AssertEquals_STRING(
    Expected := expected,
    Actual := actual,
    Message := 'Type did not return correct iec type.'
);

TEST_FINISHED();
END_METHOD

METHOD PUBLIC TestIsSigned
VAR
    _type : _ULINT(0);
    expected : STRING := 'BOOL';
    actual : STRING;
END_VAR
TEST('TestIsSigned');

AssertFalse(
	Condition := _type.IsSigned,
    Message := 'Type did not correctly identify itself as being unsigned'
);

TEST_FINISHED();
END_METHOD

METHOD PUBLIC TestMakeReferenceToFollowsReference
VAR
    _type : _ULINT(0);
	target : ULINT := 0;
    expected : ULINT := 123;
    actual : ULINT;
END_VAR
TEST('TestMakeReferenceToFollowsReference');

_type.MakeReferenceTo(target);
target := 123;

actual := _type.Value;

AssertEquals(
    Expected := expected,
    Actual := actual,
    Message := 'Value did not follow target change'
);

TEST_FINISHED();
END_METHOD

METHOD PUBLIC TestMakeReferenceToUpdatesReference
VAR
    _type : _ULINT(0);
	target : ULINT := 0;
    expected : ULINT := 123;
    actual : ULINT;
END_VAR
TEST('TestMakeReferenceToUpdatesReference');

_type.MakeReferenceTo(target);
_type.Value := 123;

actual := target;

AssertEquals(
    Expected := expected,
    Actual := actual,
    Message := 'Value did not update target'
);

TEST_FINISHED();
END_METHOD

METHOD PUBLIC TestSerializeTypeWith
VAR
    _type : _ULINT(0);
    serializer : JsonSerializer;
    expected : STRING(500) := '{"datatype":"ULINT","lowerBound":0,"upperBound":18446744073709551615,"isSigned":false}';
    actual : STRING(500);
END_VAR
TEST('TestSerializeTypeWith');

serializer.Reset();
_type.SerializeTypeWith(serializer);
serializer.TryGetSerializedData(ADR(actual), SIZEOF(actual));

AssertEquals_STRING(
    Expected := expected,
    Actual := actual,
    Message := 'Serialization of type did not return correct string.'
);

TEST_FINISHED();
END_METHOD

METHOD PUBLIC TestSerializeWith
VAR
    _type : _ULINT(32767);
    serializer : JsonSerializer;
    expected : STRING := '32767';
    actual : STRING(500);
END_VAR
TEST('TestSerializeWith');

serializer.Reset();
_type.SerializeWith(serializer);
serializer.TryGetSerializedData(ADR(actual), SIZEOF(actual));

AssertEquals_STRING(
    Expected := expected,
    Actual := actual,
    Message := 'Serialization of type data did not return correct string.'
);

TEST_FINISHED();
END_METHOD

METHOD PUBLIC TestSize
VAR
    _type : _ULINT(0);
    expected : UDINT := SIZEOF(ULINT);
    actual : UDINT;
END_VAR
TEST('TestSize');

actual := _type.Size;

AssertEquals_UDINT(
    Expected := Expected,
    Actual := actual,
    Message := 'Type did not return the correct size.'
);

TEST_FINISHED();
END_METHOD

METHOD PUBLIC TestTryDeserializeFrom
VAR
    deserializer : JsonDeserializer;
    feedback : DeserializerFeedback;
    json : STRING := '32767';
    _type : _ULINT(0);
    expected : ULINT := 32767;
    actual : ULINT;
 END_VAR
TEST('TestTryDeserializeFrom');

deserializer.Reset();
deserializer.TryLoad(json);
_type.TryDeserializeFrom(Deserializer, Feedback);

actual := _type.Value;

AssertEquals(
    Expected := expected,
    Actual := actual,
    Message := 'Type did not deserialize correctly.'
);

TEST_FINISHED();
END_METHOD

METHOD PUBLIC TestTryMakeReferenceToFollowsReference
VAR
    _type : _ULINT(0);
	target : _ULINT(0);
    expected : ULINT := 123;
    actual : ULINT;
END_VAR
TEST('TestTryMakeReferenceToFollowsReference');

_type.TryMakeReferenceTo(target);
target.Value := 123;

actual := _type.Value;

AssertEquals(
    Expected := expected,
    Actual := actual,
    Message := 'Value did not follow target change'
);

TEST_FINISHED();
END_METHOD

METHOD PUBLIC TestTryMakeReferenceToUpdatesReference
VAR
    _type : _ULINT(0);
	target : _ULINT(0);
    expected : ULINT := 123;
    actual : ULINT;
END_VAR
TEST('TestTryMakeReferenceToUpdatesReference');

_type.TryMakeReferenceTo(target);
_type.Value := 123;

actual := target.Value;

AssertEquals(
    Expected := expected,
    Actual := actual,
    Message := 'Value did not update target'
);

TEST_FINISHED();
END_METHOD

METHOD PUBLIC TestValueReturnsExpectedAfterChange
VAR
    _type : _ULINT(0);
    expected : ULINT := 32767;
    actual : ULINT;
END_VAR
TEST('TestValueReturnsExpectedAfterChange');

_type.Value := 32767;

actual := _type.Value;

AssertEquals(
    Expected := expected,
    Actual := actual,
    Message := 'Expected value not returned after change.'
);

TEST_FINISHED();
END_METHOD

METHOD PUBLIC TestValueReturnsExpectedAfterInit
VAR
    _type : _ULINT(32767);
    expected : ULINT := 32767;
    actual : ULINT;
END_VAR
TEST('TestValueReturnsExpectedAfterInit');

actual := _type.Value;

AssertEquals(
    Expected := expected,
    Actual := actual,
    Message := 'Expected value not returned after Init.'
);

TEST_FINISHED();
END_METHOD

END_FUNCTION_BLOCK

// ---- Tests/Primitives/_REAL_TestSuite.TcPOU
FUNCTION_BLOCK _REAL_TestSuite EXTENDS TcUnit.FB_TestSuite
VAR
END_VAR

TestAddress();
TestClearReference();
TestClone();
TestIecTypeReturnsExpected();
TestIsSigned();
TestMakeReferenceToFollowsReference();
TestMakeReferenceToUpdatesReference();
TestSize();
TestValueReturnsExpectedAfterInit();
TestValueReturnsExpectedAfterChange();
TestSerializeTypeWith();
TestSerializeWith();
TestTryDeserializeFrom();
TestTryMakeReferenceToFollowsReference();
TestTryMakeReferenceToUpdatesReference();

METHOD PUBLIC TestAddress
VAR
    _type : _REAL(0.0);
    notExpected : PVOID := 0;
    actual : PVOID;
END_VAR
TEST('TestAddress');

actual := _type.Address;

AssertFalse(
    Condition := (notExpected = actual),
    Message := 'Type did not return a valid address.'
);

TEST_FINISHED();
END_METHOD

METHOD PUBLIC TestClearReference
VAR
    _type : _REAL(0.0);
	target : REAL := 0.0;
    expected : REAL := 0.0;
    actual : REAL;
END_VAR
TEST('TestClearReference');

_type.MakeReferenceTo(target);
_type.ClearReference();
target := 123.4;

actual := _type.Value;

AssertEquals_REAL(
    Expected := expected,
    Actual := actual,
    Delta := REAL#0.001,
    Message := 'Value did not follow target change'
);

TEST_FINISHED();
END_METHOD

METHOD PUBLIC TestClone
VAR
    _type : _REAL(123.4);
	clone : I_Datatype;
	isValidClone : BOOL;
	compareResult : DINT;
END_VAR
TEST('TestClone');

clone := _type.Clone();

isValidClone := clone <> 0;

IF isValidClone THEN
	compareResult := memcmp(_type.Address, clone.Address, clone.Size);
END_IF

AssertTrue(
	Condition := isValidClone,
	Message := 'Clone did not produce a clone'
);

AssertEquals_DINT(
	Expected := 0,
    Actual := compareResult,
    Message := 'Clone did not return a valid clone.'
);

clone.Dispose();

TEST_FINISHED();
END_METHOD

METHOD PUBLIC TestIecTypeReturnsExpected
VAR
    _type : _REAL(0.0);
    expected : STRING := 'REAL';
    actual : STRING;
END_VAR
TEST('TestIecTypeReturnsExpected');

actual := _type.Datatype;

AssertEquals_STRING(
    Expected := expected,
    Actual := actual,
    Message := 'Type did not return correct iec type.'
);

TEST_FINISHED();
END_METHOD

METHOD PUBLIC TestIsSigned
VAR
    _type : _REAL(0);
    expected : STRING := 'BOOL';
    actual : STRING;
END_VAR
TEST('TestIsSigned');

AssertTrue(
	Condition := _type.IsSigned,
    Message := 'Type did not correctly identify itself as being signed'
);

TEST_FINISHED();
END_METHOD

METHOD PUBLIC TestMakeReferenceToFollowsReference
VAR
    _type : _REAL(0.0);
	target : REAL := 0.0;
    expected : REAL := 123.4;
    actual : REAL;
END_VAR
TEST('TestMakeReferenceToFollowsReference');

_type.MakeReferenceTo(target);
target := 123.4;

actual := _type.Value;

AssertEquals_REAL(
    Expected := expected,
    Actual := actual,
    Delta := REAL#0.001,
    Message := 'Value did not follow target change'
);

TEST_FINISHED();
END_METHOD

METHOD PUBLIC TestMakeReferenceToUpdatesReference
VAR
    _type : _REAL(0.0);
	target : REAL := 0.0;
    expected : REAL := 123.4;
    actual : REAL;
END_VAR
TEST('TestMakeReferenceToUpdatesReference');

_type.MakeReferenceTo(target);
_type.Value := 123.4;

actual := target;

AssertEquals_REAL(
    Expected := expected,
    Actual := actual,
    Delta := REAL#0.001,
    Message := 'Value did not update target'
);

TEST_FINISHED();
END_METHOD

METHOD PUBLIC TestSerializeTypeWith
VAR
    _type : _REAL(0.0);
    serializer : JsonSerializer;
    expected : STRING(500) := '{"datatype":"REAL"}';
    actual : STRING(500);
END_VAR
TEST('TestSerializeTypeWith');

serializer.Reset();
_type.SerializeTypeWith(serializer);
serializer.TryGetSerializedData(ADR(actual), SIZEOF(actual));

AssertEquals_STRING(
    Expected := expected,
    Actual := actual,
    Message := 'Serialization of type did not return correct string.'
);

TEST_FINISHED();
END_METHOD

METHOD PUBLIC TestSerializeWith
VAR
    _type : _REAL(123.4);
    serializer : JsonSerializer;
    expected : STRING := '123.40000152'; // Expected value due to the nature of floating point values defined by IEEE754.
    actual : STRING(500);
END_VAR
TEST('TestSerializeWith');

serializer.Reset();
_type.SerializeWith(serializer);
serializer.TryGetSerializedData(ADR(actual), SIZEOF(actual));

AssertEquals_STRING(
    Expected := expected,
    Actual := actual,
    Message := 'Serialization of type data did not return correct string.'
);

TEST_FINISHED();
END_METHOD

METHOD PUBLIC TestSize
VAR
    _type : _REAL(0.0);
    expected : UDINT := SIZEOF(REAL);
    actual : UDINT;
END_VAR
TEST('TestSize');

actual := _type.Size;

AssertEquals_UDINT(
    Expected := Expected,
    Actual := actual,
    Message := 'Type did not return the correct size.'
);

TEST_FINISHED();
END_METHOD

METHOD PUBLIC TestTryDeserializeFrom
VAR
    deserializer : JsonDeserializer;
    feedback : DeserializerFeedback;
    json : STRING := '123.4';
    _type : _REAL(0.0);
    expected : REAL := 123.4;
    actual : REAL;
 END_VAR
TEST('TestTryDeserializeFrom');

deserializer.Reset();
deserializer.TryLoad(json);
_type.TryDeserializeFrom(Deserializer, Feedback);

actual := _type.Value;

AssertEquals_REAL(
    Expected := expected,
    Actual := actual,
    Delta := REAL#0.001,
    Message := 'Type did not deserialize correctly.'
);

TEST_FINISHED();
END_METHOD

METHOD PUBLIC TestTryMakeReferenceToFollowsReference
VAR
    _type : _REAL(0.0);
	target : _REAL(0.0);
    expected : REAL := 123.4;
    actual : REAL;
END_VAR
TEST('TestTryMakeReferenceToFollowsReference');

_type.TryMakeReferenceTo(target);
target.Value := 123.4;

actual := _type.Value;

AssertEquals_REAL(
    Expected := expected,
    Actual := actual,
    Delta := REAL#0.001,
    Message := 'Value did not follow target change'
);

TEST_FINISHED();
END_METHOD

METHOD PUBLIC TestTryMakeReferenceToUpdatesReference
VAR
    _type : _REAL(0.0);
	target : _REAL(0.0);
    expected : REAL := 123.4;
    actual : REAL;
END_VAR
TEST('TestTryMakeReferenceToUpdatesReference');

_type.TryMakeReferenceTo(target);
_type.Value := 123.4;

actual := target.Value;

AssertEquals_REAL(
    Expected := expected,
    Actual := actual,
    Delta := REAL#0.001,
    Message := 'Value did not update target'
);

TEST_FINISHED();
END_METHOD

METHOD PUBLIC TestValueReturnsExpectedAfterChange
VAR
    _type : _REAL(0.0);
    expected : REAL := 123.4;
    actual : REAL;
END_VAR
TEST('TestValueReturnsExpectedAfterChange');

_type.Value := 123.4;

actual := _type.Value;

AssertEquals_REAL(
    Expected := expected,
    Actual := actual,
    Delta := REAL#0.001,
    Message := 'Expected value not returned after change.'
);

TEST_FINISHED();
END_METHOD

METHOD PUBLIC TestValueReturnsExpectedAfterInit
VAR
    _type : _REAL(123.4);
    expected : REAL := 123.4;
    actual : REAL;
END_VAR
TEST('TestValueReturnsExpectedAfterInit');

actual := _type.Value;

AssertEquals_REAL(
    Expected := expected,
    Actual := actual,
    Delta := REAL#0.001,
    Message := 'Expected value not returned after Init.'
);

TEST_FINISHED();
END_METHOD

END_FUNCTION_BLOCK

// ---- Tests/Primitives/_LREAL_TestSuite.TcPOU
FUNCTION_BLOCK _LREAL_TestSuite EXTENDS TcUnit.FB_TestSuite
VAR
END_VAR

TestAddress();
TestClearReference();
TestClone();
TestIecTypeReturnsExpected();
TestIsSigned();
TestMakeReferenceToFollowsReference();
TestMakeReferenceToUpdatesReference();
TestSize();
TestValueReturnsExpectedAfterInit();
TestValueReturnsExpectedAfterChange();
TestSerializeTypeWith();
TestSerializeWith();
TestTryDeserializeFrom();
TestTryMakeReferenceToFollowsReference();
TestTryMakeReferenceToUpdatesReference();

METHOD PUBLIC TestAddress
VAR
    _type : _LREAL(0.0);
    notExpected : PVOID := 0;
    actual : PVOID;
END_VAR
TEST('TestAddress');

actual := _type.Address;

AssertFalse(
    Condition := (notExpected = actual),
    Message := 'Type did not return a valid address.'
);

TEST_FINISHED();
END_METHOD

METHOD PUBLIC TestClearReference
VAR
    _type : _LREAL(0.0);
	target : LREAL := 0.0;
    expected : LREAL := 0.0;
    actual : LREAL;
END_VAR
TEST('TestClearReference');

_type.MakeReferenceTo(target);
_type.ClearReference();
target := 123.4;

actual := _type.Value;

AssertEquals_LREAL(
    Expected := expected,
    Actual := actual,
    Delta := LREAL#0.001,
    Message := 'Value did not follow target change'
);

TEST_FINISHED();
END_METHOD

METHOD PUBLIC TestClone
VAR
    _type : _LREAL(123.4);
	clone : I_Datatype;
	isValidClone : BOOL;
	compareResult : DINT;
END_VAR
TEST('TestClone');

clone := _type.Clone();

isValidClone := clone <> 0;

IF isValidClone THEN
	compareResult := memcmp(_type.Address, clone.Address, clone.Size);
END_IF

AssertTrue(
	Condition := isValidClone,
	Message := 'Clone did not produce a clone'
);

AssertEquals_DINT(
	Expected := 0,
    Actual := compareResult,
    Message := 'Clone did not return a valid clone.'
);

clone.Dispose();

TEST_FINISHED();
END_METHOD

METHOD PUBLIC TestIecTypeReturnsExpected
VAR
    _type : _LREAL(0.0);
    expected : STRING := 'LREAL';
    actual : STRING;
END_VAR
TEST('TestIecTypeReturnsExpected');

actual := _type.Datatype;

AssertEquals_STRING(
    Expected := expected,
    Actual := actual,
    Message := 'Type did not return correct iec type.'
);

TEST_FINISHED();
END_METHOD

METHOD PUBLIC TestIsSigned
VAR
    _type : _LREAL(0);
    expected : STRING := 'BOOL';
    actual : STRING;
END_VAR
TEST('TestIsSigned');

AssertTrue(
	Condition := _type.IsSigned,
    Message := 'Type did not correctly identify itself as being signed'
);

TEST_FINISHED();
END_METHOD

METHOD PUBLIC TestMakeReferenceToFollowsReference
VAR
    _type : _LREAL(0.0);
	target : LREAL := 0.0;
    expected : LREAL := 123.4;
    actual : LREAL;
END_VAR
TEST('TestMakeReferenceToFollowsReference');

_type.MakeReferenceTo(target);
target := 123.4;

actual := _type.Value;

AssertEquals_LREAL(
    Expected := expected,
    Actual := actual,
    Delta := LREAL#0.001,
    Message := 'Value did not follow target change'
);

TEST_FINISHED();
END_METHOD

METHOD PUBLIC TestMakeReferenceToUpdatesReference
VAR
    _type : _LREAL(0.0);
	target : LREAL := 0.0;
    expected : LREAL := 123.4;
    actual : LREAL;
END_VAR
TEST('TestMakeReferenceToUpdatesReference');

_type.MakeReferenceTo(target);
_type.Value := 123.4;

actual := target;

AssertEquals_LREAL(
    Expected := expected,
    Actual := actual,
    Delta := LREAL#0.001,
    Message := 'Value did not update target'
);

TEST_FINISHED();
END_METHOD

METHOD PUBLIC TestSerializeTypeWith
VAR
    _type : _LREAL(0.0);
    serializer : JsonSerializer;
    expected : STRING(500) := '{"datatype":"LREAL"}';
    actual : STRING(500);
END_VAR
TEST('TestSerializeTypeWith');

serializer.Reset();
_type.SerializeTypeWith(serializer);
serializer.TryGetSerializedData(ADR(actual), SIZEOF(actual));

AssertEquals_STRING(
    Expected := expected,
    Actual := actual,
    Message := 'Serialization of type did not return correct string.'
);

TEST_FINISHED();
END_METHOD

METHOD PUBLIC TestSerializeWith
VAR
    _type : _LREAL(123.4);
    serializer : JsonSerializer;
    expected : STRING := '123.4';
    actual : STRING(500);
END_VAR
TEST('TestSerializeWith');

serializer.Reset();
_type.SerializeWith(serializer);
serializer.TryGetSerializedData(ADR(actual), SIZEOF(actual));

AssertEquals_STRING(
    Expected := expected,
    Actual := actual,
    Message := 'Serialization of type data did not return correct string.'
);

TEST_FINISHED();
END_METHOD

METHOD PUBLIC TestSize
VAR
    _type : _LREAL(0.0);
    expected : UDINT := SIZEOF(LREAL);
    actual : UDINT;
END_VAR
TEST('TestSize');

actual := _type.Size;

AssertEquals_UDINT(
    Expected := Expected,
    Actual := actual,
    Message := 'Type did not return the correct size.'
);

TEST_FINISHED();
END_METHOD

METHOD PUBLIC TestTryDeserializeFrom
VAR
    deserializer : JsonDeserializer;
    feedback : DeserializerFeedback;
    json : STRING := '123.4';
    _type : _LREAL(0.0);
    expected : LREAL := 123.4;
    actual : LREAL;
 END_VAR
TEST('TestTryDeserializeFrom');

deserializer.Reset();
deserializer.TryLoad(json);
_type.TryDeserializeFrom(Deserializer, Feedback);

actual := _type.Value;

AssertEquals_LREAL(
    Expected := expected,
    Actual := actual,
    Delta := LREAL#0.001,
    Message := 'Type did not deserialize correctly.'
);

TEST_FINISHED();
END_METHOD

METHOD PUBLIC TestTryMakeReferenceToFollowsReference
VAR
    _type : _LREAL(0.0);
	target : _LREAL(0.0);
    expected : LREAL := 123.4;
    actual : LREAL;
END_VAR
TEST('TestTryMakeReferenceToFollowsReference');

_type.TryMakeReferenceTo(target);
target.Value := 123.4;

actual := _type.Value;

AssertEquals_LREAL(
    Expected := expected,
    Actual := actual,
    Delta := LREAL#0.001,
    Message := 'Value did not follow target change'
);

TEST_FINISHED();
END_METHOD

METHOD PUBLIC TestTryMakeReferenceToUpdatesReference
VAR
    _type : _LREAL(0.0);
	target : _LREAL(0.0);
    expected : LREAL := 123.4;
    actual : LREAL;
END_VAR
TEST('TestTryMakeReferenceToUpdatesReference');

_type.TryMakeReferenceTo(target);
_type.Value := 123.4;

actual := target.Value;

AssertEquals_LREAL(
    Expected := expected,
    Actual := actual,
    Delta := LREAL#0.001,
    Message := 'Value did not update target'
);

TEST_FINISHED();
END_METHOD

METHOD PUBLIC TestValueReturnsExpectedAfterChange
VAR
    _type : _LREAL(0.0);
    expected : LREAL := 123.4;
    actual : LREAL;
END_VAR
TEST('TestValueReturnsExpectedAfterChange');

_type.Value := 123.4;

actual := _type.Value;

AssertEquals_LREAL(
    Expected := expected,
    Actual := actual,
    Delta := LREAL#0.001,
    Message := 'Expected value not returned after change.'
);

TEST_FINISHED();
END_METHOD

METHOD PUBLIC TestValueReturnsExpectedAfterInit
VAR
    _type : _LREAL(123.4);
    expected : LREAL := 123.4;
    actual : LREAL;
END_VAR
TEST('TestValueReturnsExpectedAfterInit');

actual := _type.Value;

AssertEquals_LREAL(
    Expected := expected,
    Actual := actual,
    Delta := LREAL#0.001,
    Message := 'Expected value not returned after Init.'
);

TEST_FINISHED();
END_METHOD

END_FUNCTION_BLOCK

// ---- Tests/Primitives/_TOD_TestSuite.TcPOU
FUNCTION_BLOCK _TOD_TestSuite EXTENDS TcUnit.FB_TestSuite
VAR
END_VAR

TestAddress();
TestClearReference();
TestClone();
TestIecTypeReturnsExpected();
TestMakeReferenceToFollowsReference();
TestMakeReferenceToUpdatesReference();
TestSize();
TestValueReturnsExpectedAfterInit();
TestValueReturnsExpectedAfterChange();
TestSerializeTypeWith();
TestSerializeWith();
TestTryDeserializeFrom();
TestTryMakeReferenceToFollowsReference();
TestTryMakeReferenceToUpdatesReference();

METHOD PUBLIC TestAddress
VAR
    _type : _TOD(TOD#0:0:0);
    notExpected : PVOID := 0;
    actual : PVOID;
END_VAR
TEST('TestAddress');

actual := _type.Address;

AssertFalse(
    Condition := (notExpected = actual),
    Message := 'Type did not return a valid address.'
);

TEST_FINISHED();
END_METHOD

METHOD PUBLIC TestClearReference
VAR
    _type : _TOD(TOD#0:0:0);
	target : TOD := TOD#0:0:0;
    expected : TOD := TOD#0:0:0;
    actual : TOD;
END_VAR
TEST('TestClearReference');

_type.MakeReferenceTo(target);
_type.ClearReference();
target := TOD#12:34:56.789;

actual := _type.Value;

AssertEquals(
    Expected := expected,
    Actual := actual,
    Message := 'Value did not follow target change'
);

TEST_FINISHED();
END_METHOD

METHOD PUBLIC TestClone
VAR
    _type : _TIME_OF_DAY(TIME_OF_DAY#12:34:56.789);
	clone : I_Datatype;
	isValidClone : BOOL;
	compareResult : DINT;
END_VAR
TEST('TestClone');

clone := _type.Clone();

isValidClone := clone <> 0;

IF isValidClone THEN
	compareResult := memcmp(_type.Address, clone.Address, clone.Size);
END_IF

AssertTrue(
	Condition := isValidClone,
	Message := 'Clone did not produce a clone'
);

AssertEquals_DINT(
	Expected := 0,
    Actual := compareResult,
    Message := 'Clone did not return a valid clone.'
);

clone.Dispose();

TEST_FINISHED();
END_METHOD

METHOD PUBLIC TestIecTypeReturnsExpected
VAR
    _type : _TOD(TOD#0:0:0);
    expected : STRING := 'TOD';
    actual : STRING;
END_VAR
TEST('TestIecTypeReturnsExpected');

actual := _type.Datatype;

AssertEquals_STRING(
    Expected := expected,
    Actual := actual,
    Message := 'Type did not return correct iec type.'
);

TEST_FINISHED();
END_METHOD

METHOD PUBLIC TestMakeReferenceToFollowsReference
VAR
    _type : _TOD(TOD#0:0:0);
	target : TOD := TOD#0:0:0;
    expected : TOD := TOD#12:34:56.789;
    actual : TOD;
END_VAR
TEST('TestMakeReferenceToFollowsReference');

_type.MakeReferenceTo(target);
target := TOD#12:34:56.789;

actual := _type.Value;

AssertEquals_TIME_OF_DAY(
    Expected := expected,
    Actual := actual,
    Message := 'Value did not follow target change'
);

TEST_FINISHED();
END_METHOD

METHOD PUBLIC TestMakeReferenceToUpdatesReference
VAR
    _type : _TOD(TOD#0:0:0);
	target : TOD := TOD#0:0:0;
    expected : TOD := TOD#12:34:56.789;
    actual : TOD;
END_VAR
TEST('TestMakeReferenceToUpdatesReference');

_type.MakeReferenceTo(target);
_type.Value := TOD#12:34:56.789;

actual := target;

AssertEquals_TIME_OF_DAY(
    Expected := expected,
    Actual := actual,
    Message := 'Value did not update target'
);

TEST_FINISHED();
END_METHOD

METHOD PUBLIC TestSerializeTypeWith
VAR
    _type : _TOD(TOD#0:0:0);
    serializer : JsonSerializer;
    expected : STRING := '{"datatype":"TOD"}';
    actual : STRING(500);
END_VAR
TEST('TestSerializeTypeWith');

serializer.Reset();
_type.SerializeTypeWith(serializer);
serializer.TryGetSerializedData(ADR(actual), SIZEOF(actual));

AssertEquals_STRING(
    Expected := expected,
    Actual := actual,
    Message := 'Serialization of type did not return correct string.'
);

TEST_FINISHED();
END_METHOD

METHOD PUBLIC TestSerializeWith
VAR
    _type : _TOD(TOD#12:34:56.789);
    serializer : JsonSerializer;
    expected : STRING := '"TOD#12:34:56.789"';
    actual : STRING(500);
END_VAR
TEST('TestSerializeWith');

serializer.Reset();
_type.SerializeWith(serializer);
serializer.TryGetSerializedData(ADR(actual), SIZEOF(actual));

AssertEquals_STRING(
    Expected := expected,
    Actual := actual,
    Message := 'Serialization of type data did not return correct string.'
);

TEST_FINISHED();
END_METHOD

METHOD PUBLIC TestSize
VAR
    _type : _TOD(TOD#0:0:0);
    expected : UDINT := SIZEOF(TOD);
    actual : UDINT;
END_VAR
TEST('TestSize');

actual := _type.Size;

AssertEquals_UDINT(
    Expected := Expected,
    Actual := actual,
    Message := 'Type did not return the correct size.'
);

TEST_FINISHED();
END_METHOD

METHOD PUBLIC TestTryDeserializeFrom
VAR
    deserializer : JsonDeserializer;
    feedback : DeserializerFeedback;
    json : STRING := '"TOD#12:34:56.789"';
    _type : _TOD(TOD#0:0:0);
    expected : TOD := TOD#12:34:56.789;
    actual : TOD;
 END_VAR
TEST('TestTryDeserializeFrom');

deserializer.Reset();
deserializer.TryLoad(json);
_type.TryDeserializeFrom(Deserializer, Feedback);

actual := _type.Value;

AssertEquals_TIME_OF_DAY(
    Expected := expected,
    Actual := actual,
    Message := 'Type did not deserialize correctly.'
);

TEST_FINISHED();
END_METHOD

METHOD PUBLIC TestTryMakeReferenceToFollowsReference
VAR
    _type : _TOD(TOD#0:0:0);
	target : _TOD(TOD#0:0:0);
    expected : TOD := TOD#12:34:56.789;
    actual : TOD;
END_VAR
TEST('TestTryMakeReferenceToFollowsReference');

_type.TryMakeReferenceTo(target);
target.Value := TOD#12:34:56.789;

actual := _type.Value;

AssertEquals_TIME_OF_DAY(
    Expected := expected,
    Actual := actual,
    Message := 'Value did not follow target change'
);

TEST_FINISHED();
END_METHOD

METHOD PUBLIC TestTryMakeReferenceToUpdatesReference
VAR
    _type : _TOD(TOD#0:0:0);
	target : _TOD(TOD#0:0:0);
    expected : TOD := TOD#12:34:56.789;
    actual : TOD;
END_VAR
TEST('TestTryMakeReferenceToUpdatesReference');

_type.TryMakeReferenceTo(target);
_type.Value := TOD#12:34:56.789;

actual := target.Value;

AssertEquals_TIME_OF_DAY(
    Expected := expected,
    Actual := actual,
    Message := 'Value did not update target'
);

TEST_FINISHED();
END_METHOD

METHOD PUBLIC TestValueReturnsExpectedAfterChange
VAR
    _type : _TOD(TOD#0:0:0);
    expected : TOD := TOD#12:34:56.789;
    actual : TOD;
END_VAR
TEST('TestValueReturnsExpectedAfterChange');

_type.Value := TOD#12:34:56.789;

actual := _type.Value;

AssertEquals_TIME_OF_DAY(
    Expected := expected,
    Actual := actual,
    Message := 'Expected value not returned after change.'
);

TEST_FINISHED();
END_METHOD

METHOD PUBLIC TestValueReturnsExpectedAfterInit
VAR
    _type : _TOD(TOD#12:34:56.789);
    expected : TOD := TOD#12:34:56.789;
    actual : TOD;
END_VAR
TEST('TestValueReturnsExpectedAfterInit');

actual := _type.Value;

AssertEquals_TIME_OF_DAY(
    Expected := expected,
    Actual := actual,
    Message := 'Expected value not returned after Init.'
);

TEST_FINISHED();
END_METHOD

END_FUNCTION_BLOCK

// ---- Tests/Primitives/_TIME_OF_DAY_TestSuite.TcPOU
FUNCTION_BLOCK _TIME_OF_DAY_TestSuite EXTENDS TcUnit.FB_TestSuite
VAR
END_VAR

TestAddress();
TestClearReference();
TestClone();
TestIecTypeReturnsExpected();
TestMakeReferenceToFollowsReference();
TestMakeReferenceToUpdatesReference();
TestSize();
TestValueReturnsExpectedAfterInit();
TestValueReturnsExpectedAfterChange();
TestSerializeTypeWith();
TestSerializeWith();
TestTryDeserializeFrom();
TestTryMakeReferenceToFollowsReference();
TestTryMakeReferenceToUpdatesReference();

METHOD PUBLIC TestAddress
VAR
    _type : _TIME_OF_DAY(TIME_OF_DAY#0:0:0);
    notExpected : PVOID := 0;
    actual : PVOID;
END_VAR
TEST('TestAddress');

actual := _type.Address;

AssertFalse(
    Condition := (notExpected = actual),
    Message := 'Type did not return a valid address.'
);

TEST_FINISHED();
END_METHOD

METHOD PUBLIC TestClearReference
VAR
    _type : _TIME_OF_DAY(TIME_OF_DAY#0:0:0);
	target : TIME_OF_DAY := TIME_OF_DAY#0:0:0;
    expected : TIME_OF_DAY := TIME_OF_DAY#0:0:0;
    actual : TIME_OF_DAY;
END_VAR
TEST('TestClearReference');

_type.MakeReferenceTo(target);
_type.ClearReference();
target := TIME_OF_DAY#12:34:56.789;

actual := _type.Value;

AssertEquals(
    Expected := expected,
    Actual := actual,
    Message := 'Value did not follow target change'
);

TEST_FINISHED();
END_METHOD

METHOD PUBLIC TestClone
VAR
    _type : _TIME_OF_DAY(TIME_OF_DAY#12:34:56.789);
	clone : I_Datatype;
	isValidClone : BOOL;
	compareResult : DINT;
END_VAR
TEST('TestClone');

clone := _type.Clone();

isValidClone := clone <> 0;

IF isValidClone THEN
	compareResult := memcmp(_type.Address, clone.Address, clone.Size);
END_IF

AssertTrue(
	Condition := isValidClone,
	Message := 'Clone did not produce a clone'
);

AssertEquals_DINT(
	Expected := 0,
    Actual := compareResult,
    Message := 'Clone did not return a valid clone.'
);

clone.Dispose();

TEST_FINISHED();
END_METHOD

METHOD PUBLIC TestIecTypeReturnsExpected
VAR
    _type : _TIME_OF_DAY(TIME_OF_DAY#0:0:0);
    expected : STRING := 'TIME_OF_DAY';
    actual : STRING;
END_VAR
TEST('TestIecTypeReturnsExpected');

actual := _type.Datatype;

AssertEquals_STRING(
    Expected := expected,
    Actual := actual,
    Message := 'Type did not return correct iec type.'
);

TEST_FINISHED();
END_METHOD

METHOD PUBLIC TestMakeReferenceToFollowsReference
VAR
    _type : _TIME_OF_DAY(TIME_OF_DAY#0:0:0);
	target : TIME_OF_DAY := TIME_OF_DAY#0:0:0;
    expected : TIME_OF_DAY := TIME_OF_DAY#12:34:56.789;
    actual : TIME_OF_DAY;
END_VAR
TEST('TestMakeReferenceToFollowsReference');

_type.MakeReferenceTo(target);
target := TIME_OF_DAY#12:34:56.789;;

actual := _type.Value;

AssertEquals_TIME_OF_DAY(
    Expected := expected,
    Actual := actual,
    Message := 'Value did not follow target change'
);

TEST_FINISHED();
END_METHOD

METHOD PUBLIC TestMakeReferenceToUpdatesReference
VAR
    _type : _TIME_OF_DAY(TIME_OF_DAY#0:0:0);
	target : TIME_OF_DAY := TIME_OF_DAY#0:0:0;
    expected : TIME_OF_DAY := TIME_OF_DAY#12:34:56.789;
    actual : TIME_OF_DAY;
END_VAR
TEST('TestMakeReferenceToUpdatesReference');

_type.MakeReferenceTo(target);
_type.Value := TIME_OF_DAY#12:34:56.789;

actual := target;

AssertEquals_TIME_OF_DAY(
    Expected := expected,
    Actual := actual,
    Message := 'Value did not update target'
);

TEST_FINISHED();
END_METHOD

METHOD PUBLIC TestSerializeTypeWith
VAR
    _type : _TIME_OF_DAY(TIME_OF_DAY#0:0:0);
    serializer : JsonSerializer;
    expected : STRING := '{"datatype":"TIME_OF_DAY"}';
    actual : STRING(500);
END_VAR
TEST('TestSerializeTypeWith');

serializer.Reset();
_type.SerializeTypeWith(serializer);
serializer.TryGetSerializedData(ADR(actual), SIZEOF(actual));

AssertEquals_STRING(
    Expected := expected,
    Actual := actual,
    Message := 'Serialization of type did not return correct string.'
);

TEST_FINISHED();
END_METHOD

METHOD PUBLIC TestSerializeWith
VAR
    _type : _TIME_OF_DAY(TIME_OF_DAY#12:34:56.789);
    serializer : JsonSerializer;
    expected : STRING := '"TOD#12:34:56.789"';
    actual : STRING(500);
END_VAR
TEST('TestSerializeWith');

serializer.Reset();
_type.SerializeWith(serializer);
serializer.TryGetSerializedData(ADR(actual), SIZEOF(actual));

AssertEquals_STRING(
    Expected := expected,
    Actual := actual,
    Message := 'Serialization of type data did not return correct string.'
);

TEST_FINISHED();
END_METHOD

METHOD PUBLIC TestSize
VAR
    _type : _TIME_OF_DAY(TIME_OF_DAY#0:0:0);
    expected : UDINT := SIZEOF(TIME_OF_DAY);
    actual : UDINT;
END_VAR
TEST('TestSize');

actual := _type.Size;

AssertEquals_UDINT(
    Expected := Expected,
    Actual := actual,
    Message := 'Type did not return the correct size.'
);

TEST_FINISHED();
END_METHOD

METHOD PUBLIC TestTryDeserializeFrom
VAR
    deserializer : JsonDeserializer;
    feedback : DeserializerFeedback;
    json : STRING := '"TIME_OF_DAY#12:34:56.789"';
    _type : _TIME_OF_DAY(TIME_OF_DAY#0:0:0);
    expected : TIME_OF_DAY := TIME_OF_DAY#12:34:56.789;
    actual : TIME_OF_DAY;
 END_VAR
TEST('TestTryDeserializeFrom');

deserializer.Reset();
deserializer.TryLoad(json);
_type.TryDeserializeFrom(Deserializer, Feedback);

actual := _type.Value;

AssertEquals_TIME_OF_DAY(
    Expected := expected,
    Actual := actual,
    Message := 'Type did not deserialize correctly.'
);

TEST_FINISHED();
END_METHOD

METHOD PUBLIC TestTryMakeReferenceToFollowsReference
VAR
    _type : _TIME_OF_DAY(TIME_OF_DAY#0:0:0);
	target : _TIME_OF_DAY(TIME_OF_DAY#0:0:0);
    expected : TIME_OF_DAY := TIME_OF_DAY#12:34:56.789;
    actual : TIME_OF_DAY;
END_VAR
TEST('TestTryMakeReferenceToFollowsReference');

_type.TryMakeReferenceTo(target);
target.Value := TIME_OF_DAY#12:34:56.789;

actual := _type.Value;

AssertEquals_TIME_OF_DAY(
    Expected := expected,
    Actual := actual,
    Message := 'Value did not follow target change'
);

TEST_FINISHED();
END_METHOD

METHOD PUBLIC TestTryMakeReferenceToUpdatesReference
VAR
    _type : _TIME_OF_DAY(TIME_OF_DAY#0:0:0);
	target : _TIME_OF_DAY(TIME_OF_DAY#0:0:0);
    expected : TIME_OF_DAY := TIME_OF_DAY#12:34:56.789;
    actual : TIME_OF_DAY;
END_VAR
TEST('TestTryMakeReferenceToUpdatesReference');

_type.TryMakeReferenceTo(target);
_type.Value := TIME_OF_DAY#12:34:56.789;

actual := target.Value;

AssertEquals_TIME_OF_DAY(
    Expected := expected,
    Actual := actual,
    Message := 'Value did not update target'
);

TEST_FINISHED();
END_METHOD

METHOD PUBLIC TestValueReturnsExpectedAfterChange
VAR
    _type : _TIME_OF_DAY(TIME_OF_DAY#0:0:0);
    expected : TIME_OF_DAY := TIME_OF_DAY#12:34:56.789;
    actual : TIME_OF_DAY;
END_VAR
TEST('TestValueReturnsExpectedAfterChange');

_type.Value := TIME_OF_DAY#12:34:56.789;

actual := _type.Value;

AssertEquals_TIME_OF_DAY(
    Expected := expected,
    Actual := actual,
    Message := 'Expected value not returned after change.'
);

TEST_FINISHED();
END_METHOD

METHOD PUBLIC TestValueReturnsExpectedAfterInit
VAR
    _type : _TIME_OF_DAY(TIME_OF_DAY#12:34:56.789);
    expected : TIME_OF_DAY := TIME_OF_DAY#12:34:56.789;
    actual : TIME_OF_DAY;
END_VAR
TEST('TestValueReturnsExpectedAfterInit');

actual := _type.Value;

AssertEquals_TIME_OF_DAY(
    Expected := expected,
    Actual := actual,
    Message := 'Expected value not returned after Init.'
);

TEST_FINISHED();
END_METHOD

END_FUNCTION_BLOCK

// ---- Tests/Primitives/_DT_TestSuite.TcPOU
FUNCTION_BLOCK _DT_TestSuite EXTENDS TcUnit.FB_TestSuite
VAR
END_VAR

TestAddress();
TestClearReference();
TestClone();
TestIecTypeReturnsExpected();
TestMakeReferenceToFollowsReference();
TestMakeReferenceToUpdatesReference();
TestSize();
TestValueReturnsExpectedAfterInit();
TestValueReturnsExpectedAfterChange();
TestSerializeTypeWith();
TestSerializeWith();
TestTryDeserializeFrom();
TestTryMakeReferenceToFollowsReference();
TestTryMakeReferenceToUpdatesReference();

METHOD PUBLIC TestAddress
VAR
    _type : _DT(DT#1970-1-1-0:0:0);
    notExpected : PVOID := 0;
    actual : PVOID;
END_VAR
TEST('TestAddress');

actual := _type.Address;

AssertFalse(
    Condition := (notExpected = actual),
    Message := 'Type did not return a valid address.'
);

TEST_FINISHED();
END_METHOD

METHOD PUBLIC TestClearReference
VAR
    _type : _DT(DT#1970-1-1-0:0:0);
	target : DT := DT#1970-1-1-0:0:0;
    expected : DT := DT#1970-1-1-0:0:0;
    actual : DT;
END_VAR
TEST('TestClearReference');

_type.MakeReferenceTo(target);
_type.ClearReference();
target := DT#2024-12-31-12:34:56;

actual := _type.Value;

AssertEquals(
    Expected := expected,
    Actual := actual,
    Message := 'Value did not follow target change'
);

TEST_FINISHED();
END_METHOD

METHOD PUBLIC TestClone
VAR
    _type : _DT(DT#2024-12-31-12:34:56);
	clone : I_Datatype;
	isValidClone : BOOL;
	compareResult : DINT;
END_VAR
TEST('TestClone');

clone := _type.Clone();

isValidClone := clone <> 0;

IF isValidClone THEN
	compareResult := memcmp(_type.Address, clone.Address, clone.Size);
END_IF

AssertTrue(
	Condition := isValidClone,
	Message := 'Clone did not produce a clone'
);

AssertEquals_DINT(
	Expected := 0,
    Actual := compareResult,
    Message := 'Clone did not return a valid clone.'
);

clone.Dispose();

TEST_FINISHED();
END_METHOD

METHOD PUBLIC TestIecTypeReturnsExpected
VAR
    _type : _DT(DT#2024-12-31-12:34:56);
    expected : STRING := 'DT';
    actual : STRING;
END_VAR
TEST('TestIecTypeReturnsExpected');

actual := _type.Datatype;

AssertEquals_STRING(
    Expected := expected,
    Actual := actual,
    Message := 'Type did not return correct iec type.'
);

TEST_FINISHED();
END_METHOD

METHOD PUBLIC TestMakeReferenceToFollowsReference
VAR
    _type : _DT(DT#1970-1-1-0:0:0);
	target : DT := DT#1970-1-1-0:0:0;
    expected : DT := DT#2024-12-31-12:34:56;
    actual : DT;
END_VAR
TEST('TestMakeReferenceToFollowsReference');

_type.MakeReferenceTo(target);
target := DT#2024-12-31-12:34:56;

actual := _type.Value;

AssertEquals_DATE_AND_TIME(
    Expected := expected,
    Actual := actual,
    Message := 'Value did not follow target change'
);

TEST_FINISHED();
END_METHOD

METHOD PUBLIC TestMakeReferenceToUpdatesReference
VAR
    _type : _DT(DT#1970-1-1-0:0:0);
	target : DT := DT#1970-1-1-0:0:0;
    expected : DT := DT#2024-12-31-12:34:56;
    actual : DT;
END_VAR
TEST('TestMakeReferenceToUpdatesReference');

_type.MakeReferenceTo(target);
_type.Value := DT#2024-12-31-12:34:56;

actual := target;

AssertEquals_DATE_AND_TIME(
    Expected := expected,
    Actual := actual,
    Message := 'Value did not update target'
);

TEST_FINISHED();
END_METHOD

METHOD PUBLIC TestSerializeTypeWith
VAR
    _type : _DT(DT#2024-12-31-12:34:56);
    serializer : JsonSerializer;
    expected : STRING := '{"datatype":"DT"}';
    actual : STRING(500);
END_VAR
TEST('TestSerializeTypeWith');

serializer.Reset();
_type.SerializeTypeWith(serializer);
serializer.TryGetSerializedData(ADR(actual), SIZEOF(actual));

AssertEquals_STRING(
    Expected := expected,
    Actual := actual,
    Message := 'Serialization of type did not return correct string.'
);

TEST_FINISHED();
END_METHOD

METHOD PUBLIC TestSerializeWith
VAR
    _type : _DT(DT#2024-12-31-12:34:56);
    serializer : JsonSerializer;
    expected : STRING := '"2024-12-31T12:34:56"';
    actual : STRING(500);
END_VAR
TEST('TestSerializeWith');

serializer.Reset();
_type.SerializeWith(serializer);
serializer.TryGetSerializedData(ADR(actual), SIZEOF(actual));

AssertEquals_STRING(
    Expected := expected,
    Actual := actual,
    Message := 'Serialization of type data did not return correct string.'
);

TEST_FINISHED();
END_METHOD

METHOD PUBLIC TestSize
VAR
    _type : _DT(DT#1970-1-1-0:0:0);
    expected : UDINT := SIZEOF(DT);
    actual : UDINT;
END_VAR
TEST('TestSize');

actual := _type.Size;

AssertEquals_UDINT(
    Expected := Expected,
    Actual := actual,
    Message := 'Type did not return the correct size.'
);

TEST_FINISHED();
END_METHOD

METHOD PUBLIC TestTryDeserializeFrom
VAR
    deserializer : JsonDeserializer;
    feedback : DeserializerFeedback;
    json : STRING := '"2024-12-31T12:34:56"';
    _type : _DT(DT#1970-1-1-0:0:0);
    expected : DT := DT#2024-12-31-12:34:56;
    actual : DT;
 END_VAR
TEST('TestTryDeserializeFrom');

deserializer.Reset();
deserializer.TryLoad(json);
_type.TryDeserializeFrom(Deserializer, Feedback);

actual := _type.Value;

AssertEquals_DATE_AND_TIME(
    Expected := expected,
    Actual := actual,
    Message := 'Type did not deserialize correctly.'
);

TEST_FINISHED();
END_METHOD

METHOD PUBLIC TestTryMakeReferenceToFollowsReference
VAR
    _type : _DT(DT#1970-1-1-0:0:0);
	target : _DT(DT#1970-1-1-0:0:0);
    expected : DT := DT#2024-12-31-12:34:56;
    actual : DT;
END_VAR
TEST('TestTryMakeReferenceToFollowsReference');

_type.TryMakeReferenceTo(target);
target.Value := DT#2024-12-31-12:34:56;

actual := _type.Value;

AssertEquals_DATE_AND_TIME(
    Expected := expected,
    Actual := actual,
    Message := 'Value did not follow target change'
);

TEST_FINISHED();
END_METHOD

METHOD PUBLIC TestTryMakeReferenceToUpdatesReference
VAR
    _type : _DT(DT#1970-1-1-0:0:0);
	target : _DT(DT#1970-1-1-0:0:0);
    expected : DT := DT#2024-12-31-12:34:56;
    actual : DT;
END_VAR
TEST('TestTryMakeReferenceToUpdatesReference');

_type.TryMakeReferenceTo(target);
_type.Value := DT#2024-12-31-12:34:56;

actual := target.Value;

AssertEquals_DATE_AND_TIME(
    Expected := expected,
    Actual := actual,
    Message := 'Value did not update target'
);

TEST_FINISHED();
END_METHOD

METHOD PUBLIC TestValueReturnsExpectedAfterChange
VAR
    _type : _DT(DT#1970-1-1-0:0:0);
    expected : DT := DT#2024-12-31-12:34:56;
    actual : DT;
END_VAR
TEST('TestValueReturnsExpectedAfterChange');

_type.Value := DT#2024-12-31-12:34:56;

actual := _type.Value;

AssertEquals_DATE_AND_TIME(
    Expected := expected,
    Actual := actual,
    Message := 'Expected value not returned after change.'
);

TEST_FINISHED();
END_METHOD

METHOD PUBLIC TestValueReturnsExpectedAfterInit
VAR
    _type : _DT(DT#2024-12-31-12:34:56);
    expected : DT := DT#2024-12-31-12:34:56;
    actual : DT;
END_VAR
TEST('TestValueReturnsExpectedAfterInit');

actual := _type.Value;

AssertEquals_DATE_AND_TIME(
    Expected := expected,
    Actual := actual,
    Message := 'Expected value not returned after Init.'
);

TEST_FINISHED();
END_METHOD

END_FUNCTION_BLOCK

// ---- Tests/Primitives/_STRING_TestSuite.TcPOU
FUNCTION_BLOCK _STRING_TestSuite EXTENDS TcUnit.FB_TestSuite
VAR
END_VAR

TestAddress();
TestClearReference();
TestClone();
TestIecTypeReturnsExpected();
TestMakeReferenceToFollowsReference();
TestMakeReferenceToUpdatesReference();
TestSize();
TestValueReturnsExpectedAfterInit();
TestValueReturnsExpectedAfterChange();
TestSerializeTypeWith();
TestSerializeWith();
TestTryDeserializeFrom();
TestTryMakeReferenceToFollowsReference();
TestTryMakeReferenceToUpdatesReference();

METHOD PUBLIC TestAddress
VAR
    _type : _STRING('');
    notExpected : PVOID := 0;
    actual : PVOID;
END_VAR
TEST('TestAddress');

actual := _type.Address;

AssertFalse(
    Condition := (notExpected = actual),
    Message := 'Type did not return a valid address.'
);

TEST_FINISHED();
END_METHOD

METHOD PUBLIC TestClearReference
VAR
    _type : _STRING('');
	target : T_MaxString := '';
    expected : T_MaxString := '';
    actual : T_MaxString;
END_VAR
TEST('TestClearReference');

_type.MakeReferenceTo(target);
_type.ClearReference();
target := '123';

actual := _type.Value;

AssertEquals_STRING(
    Expected := expected,
    Actual := actual,
    Message := 'Value did not follow target change'
);

TEST_FINISHED();
END_METHOD

METHOD PUBLIC TestClone
VAR
    _type : _STRING('123');
	clone : I_Datatype;
	isValidClone : BOOL;
	compareResult : DINT;
END_VAR
TEST('TestClone');

clone := _type.Clone();

isValidClone := clone <> 0;

IF isValidClone THEN
	compareResult := memcmp(_type.Address, clone.Address, clone.Size);
END_IF

AssertTrue(
	Condition := isValidClone,
	Message := 'Clone did not produce a clone'
);

AssertEquals_DINT(
	Expected := 0,
    Actual := compareResult,
    Message := 'Clone did not return a valid clone.'
);

clone.Dispose();

TEST_FINISHED();
END_METHOD

METHOD PUBLIC TestIecTypeReturnsExpected
VAR
    _type : _STRING('');
    expected : STRING := 'STRING';
    actual : STRING;
END_VAR
TEST('TestIecTypeReturnsExpected');

actual := _type.Datatype;

AssertEquals_STRING(
    Expected := expected,
    Actual := actual,
    Message := 'Type did not return correct iec type.'
);

TEST_FINISHED();
END_METHOD

METHOD PUBLIC TestMakeReferenceToFollowsReference
VAR
    _type : _STRING('');
	target : T_MaxString := '';
    expected : T_MaxString := '123';
    actual : T_MaxString;
END_VAR
TEST('TestMakeReferenceToFollowsReference');

_type.MakeReferenceTo(target);
target := '123';

actual := _type.Value;

AssertEquals_STRING(
    Expected := expected,
    Actual := actual,
    Message := 'Value did not follow target change'
);

TEST_FINISHED();
END_METHOD

METHOD PUBLIC TestMakeReferenceToUpdatesReference
VAR
    _type : _STRING('');
	target : T_MaxString := '';
    expected : T_MaxString := '123';
    actual : T_MaxString;
END_VAR
TEST('TestMakeReferenceToUpdatesReference');

_type.MakeReferenceTo(target);
_type.Value := '123';

actual := target;

AssertEquals_STRING(
    Expected := expected,
    Actual := actual,
    Message := 'Value did not update target'
);

TEST_FINISHED();
END_METHOD

METHOD PUBLIC TestSerializeTypeWith
VAR
    _type : _STRING('');
    serializer : JsonSerializer;
    expected : STRING := '{"datatype":"STRING"}';
    actual : STRING(500);
END_VAR
TEST('TestSerializeTypeWith');

serializer.Reset();
_type.SerializeTypeWith(serializer);
serializer.TryGetSerializedData(ADR(actual), SIZEOF(actual));

AssertEquals_STRING(
    Expected := expected,
    Actual := actual,
    Message := 'Serialization of type did not return correct string.'
);

TEST_FINISHED();
END_METHOD

METHOD PUBLIC TestSerializeWith
VAR
    _type : _STRING('abcdefghijklmnopqrstuvwxyzABCDEFGHIJKLMNOPQRSTUVWXYZ01234567890');
    serializer : JsonSerializer;
    expected : STRING := '"abcdefghijklmnopqrstuvwxyzABCDEFGHIJKLMNOPQRSTUVWXYZ01234567890"';
    actual : STRING(500);
END_VAR
TEST('TestSerializeWith');

serializer.Reset();
_type.SerializeWith(serializer);
serializer.TryGetSerializedData(ADR(actual), SIZEOF(actual));

AssertEquals_STRING(
    Expected := expected,
    Actual := actual,
    Message := 'Serialization of type data did not return correct string.'
);

TEST_FINISHED();
END_METHOD

METHOD PUBLIC TestSize
VAR
    _type : _STRING('');
    expected : UDINT := SIZEOF(T_MaxString);
    actual : UDINT;
END_VAR
TEST('TestSize');

actual := _type.Size;

AssertEquals_UDINT(
    Expected := Expected,
    Actual := actual,
    Message := 'Type did not return the correct size.'
);

TEST_FINISHED();
END_METHOD

METHOD PUBLIC TestTryDeserializeFrom
VAR
    deserializer : JsonDeserializer;
    feedback : DeserializerFeedback;
    json : STRING := '"abcdefghijklmnopqrstuvwxyzABCDEFGHIJKLMNOPQRSTUVWXYZ01234567890"';
    _type : _STRING('');
    expected : T_MaxString := 'abcdefghijklmnopqrstuvwxyzABCDEFGHIJKLMNOPQRSTUVWXYZ01234567890';
    actual : T_MaxString;
 END_VAR
TEST('TestTryDeserializeFrom');

deserializer.Reset();
deserializer.TryLoad(json);
_type.TryDeserializeFrom(Deserializer, Feedback);

actual := _type.Value;

AssertEquals_STRING(
    Expected := expected,
    Actual := actual,
    Message := 'Type did not deserialize correctly.'
);

TEST_FINISHED();
END_METHOD

METHOD PUBLIC TestTryMakeReferenceToFollowsReference
VAR
    _type : _STRING('');
	target : _STRING('');
    expected : T_MaxString := '123';
    actual : T_MaxString;
END_VAR
TEST('TestTryMakeReferenceToFollowsReference');

_type.TryMakeReferenceTo(target);
target.Value := '123';

actual := _type.Value;

AssertEquals_STRING(
    Expected := expected,
    Actual := actual,
    Message := 'Value did not follow target change'
);

TEST_FINISHED();
END_METHOD

METHOD PUBLIC TestTryMakeReferenceToUpdatesReference
VAR
    _type : _STRING('');
	target : _STRING('');
    expected : T_MaxString := '123';
    actual : T_MaxString;
END_VAR
TEST('TestTryMakeReferenceToUpdatesReference');

_type.TryMakeReferenceTo(target);
_type.Value := '123';

actual := target.Value;

AssertEquals_STRING(
    Expected := expected,
    Actual := actual,
    Message := 'Value did not update target'
);

TEST_FINISHED();
END_METHOD

METHOD PUBLIC TestValueReturnsExpectedAfterChange
VAR
    _type : _STRING('');
    expected : T_MaxString := '123';
    actual : T_MaxString;
END_VAR
TEST('TestValueReturnsExpectedAfterChange');

_type.Value := '123';

actual := _type.Value;

AssertEquals_STRING(
    Expected := expected,
    Actual := actual,
    Message := 'Expected value not returned after change.'
);

TEST_FINISHED();
END_METHOD

METHOD PUBLIC TestValueReturnsExpectedAfterInit
VAR
    _type : _STRING('123');
    expected : T_MaxString := '123';
    actual : T_MaxString;
END_VAR
TEST('TestValueReturnsExpectedAfterInit');

actual := _type.Value;

AssertEquals_STRING(
    Expected := expected,
    Actual := actual,
    Message := 'Expected value not returned after Init.'
);

TEST_FINISHED();
END_METHOD

END_FUNCTION_BLOCK

// ---- Tests/Structs/_TIMESTRUCT_TestSuite.TcPOU
FUNCTION_BLOCK _TIMESTRUCT_TestSuite EXTENDS TcUnit.FB_TestSuite
VAR
END_VAR

TestAddress();
TestClearReference();
TestClone();
TestIecTypeReturnsExpected();
TestMakeReferenceToFollowsReference();
TestMakeReferenceToUpdatesReference();
TestSize();
TestValueReturnsExpectedAfterChange();
TestSerializeTypeWith();
TestSerializeWith();
TestTryDeserializeFrom();
TestTryMakeReferenceToFollowsReference();
TestTryMakeReferenceToUpdatesReference();

METHOD PUBLIC TestAddress
VAR
    _type : _TIMESTRUCT;
    notExpected : PVOID := 0;
    actual : PVOID;
END_VAR
TEST('TestAddress');

actual := _type.Address;

AssertFalse(
    Condition := (notExpected = actual),
    Message := 'Type did not return a valid address.'
);

TEST_FINISHED();
END_METHOD

METHOD PUBLIC TestClearReference
VAR
    _type : _TIMESTRUCT;
	target : TIMESTRUCT;
    expected : TIMESTRUCT;
    actual : TIMESTRUCT;
END_VAR
TEST('TestClearReference');

_type.MakeReferenceTo(target);
_type.ClearReference();
target.wDay := 2;

actual := _type.Value;

AssertEquals(
    Expected := expected,
    Actual := actual,
    Message := 'Value did not follow target change'
);

TEST_FINISHED();
END_METHOD

METHOD PUBLIC TestClone
VAR
    _type : _TIMESTRUCT;
	clone : I_Datatype;
	isValidClone : BOOL;
	compareResult : DINT;
END_VAR
TEST('TestClone');

clone := _type.Clone();

isValidClone := clone <> 0;

IF isValidClone THEN
	compareResult := memcmp(_type.Address, clone.Address, clone.Size);
END_IF

AssertTrue(
	Condition := isValidClone,
	Message := 'Clone did not produce a clone'
);

AssertEquals_DINT(
	Expected := 0,
    Actual := compareResult,
    Message := 'Clone did not return a valid clone.'
);

clone.Dispose();

TEST_FINISHED();
END_METHOD

METHOD PUBLIC TestIdentifierReturnsExpected
VAR
    _type : _HRESULT(S_OK);
    expected : STRING := 'TIMESTRUCT';
    actual : STRING;
END_VAR
TEST('TestIdentifierReturnsExpected');

actual := _type.Identifier;

AssertEquals_STRING(
    Expected := expected,
    Actual := actual,
    Message := 'Type did not return correct iec type.'
);

TEST_FINISHED();
END_METHOD

METHOD PUBLIC TestIecTypeReturnsExpected
VAR
    _type : _TIMESTRUCT;
    expected : STRING := 'STRUCT';
    actual : STRING;
END_VAR
TEST('TestIecTypeReturnsExpected');

actual := _type.Datatype;

AssertEquals_STRING(
    Expected := expected,
    Actual := actual,
    Message := 'Type did not return correct iec type.'
);

TEST_FINISHED();
END_METHOD

METHOD PUBLIC TestMakeReferenceToFollowsReference
VAR
    _type : _TIMESTRUCT;
	target : TIMESTRUCT;
    expected : TIMESTRUCT := (wDay := 2);
    actual : TIMESTRUCT;
END_VAR
TEST('TestMakeReferenceToFollowsReference');

_type.MakeReferenceTo(target);
target.wDay := 2;

actual := _type.Value;

AssertEquals(
    Expected := expected,
    Actual := actual,
    Message := 'Value did not follow target change'
);

TEST_FINISHED();
END_METHOD

METHOD PUBLIC TestMakeReferenceToUpdatesReference
VAR
    _type : _TIMESTRUCT;
	target : TIMESTRUCT;
    expected : TIMESTRUCT := (wDay := 2);
    actual : TIMESTRUCT;
END_VAR
TEST('TestMakeReferenceToUpdatesReference');

_type.MakeReferenceTo(target);
_type.wDay.Value := 2;

actual := target;

AssertEquals(
    Expected := expected,
    Actual := actual,
    Message := 'Value did not update target'
);

TEST_FINISHED();
END_METHOD

METHOD PUBLIC TestSerializeTypeWith
VAR
    _type : _TIMESTRUCT;
    serializer : JsonSerializer;
    expected : STRING(1000) := '{"datatype":"STRUCT","identifier":"TIMESTRUCT","members":{"wDay":{"datatype":"WORD","lowerBound":0,"upperBound":65535,"isSigned":false},"wDayOfWeek":{"datatype":"WORD","lowerBound":0,"upperBound":65535,"isSigned":false},"wHour":{"datatype":"WORD","lowerBound":0,"upperBound":65535,"isSigned":false},"wMilliseconds":{"datatype":"WORD","lowerBound":0,"upperBound":65535,"isSigned":false},"wMinute":{"datatype":"WORD","lowerBound":0,"upperBound":65535,"isSigned":false},"wMonth":{"datatype":"WORD","lowerBound":0,"upperBound":65535,"isSigned":false},"wSecond":{"datatype":"WORD","lowerBound":0,"upperBound":65535,"isSigned":false},"wYear":{"datatype":"WORD","lowerBound":0,"upperBound":65535,"isSigned":false}}}';
    actual : STRING(1000);
END_VAR
TEST('TestSerializeTypeWith');

serializer.Reset();
_type.SerializeTypeWith(serializer);
serializer.TryGetSerializedData(ADR(actual), SIZEOF(actual));

AssertEquals_STRING(
    Expected := expected,
    Actual := actual,
    Message := 'Serialization of type did not return correct string.'
);

TEST_FINISHED();
END_METHOD

METHOD PUBLIC TestSerializeWith
VAR
    _type : _TIMESTRUCT;
    serializer : JsonSerializer;
    expected : STRING(500) := '{"wDay":3,"wDayOfWeek":2,"wHour":4,"wMilliseconds":7,"wMinute":5,"wMonth":1,"wSecond":6,"wYear":2000}';
    actual : STRING(500);
END_VAR
TEST('TestSerializeWith');

_type.wYear.Value := 2000;
_type.wMonth.Value := 1;
_type.wDayOfWeek.Value := 2;
_type.wDay.Value := 3;
_type.wHour.Value := 4;
_type.wMinute.Value := 5;
_type.wSecond.Value := 6;
_type.wMilliseconds.Value := 7;

serializer.Reset();
_type.SerializeWith(serializer);
serializer.TryGetSerializedData(ADR(actual), SIZEOF(actual));

AssertEquals_STRING(
    Expected := expected,
    Actual := actual,
    Message := 'Serialization of type data did not return correct string.'
);

TEST_FINISHED();
END_METHOD

METHOD PUBLIC TestSize
VAR
    _type : _TIMESTRUCT;
    expected : UDINT := SIZEOF(TIMESTRUCT);
    actual : UDINT;
END_VAR
TEST('TestSize');

actual := _type.Size;

AssertEquals_UDINT(
    Expected := Expected,
    Actual := actual,
    Message := 'Type did not return the correct size.'
);

TEST_FINISHED();
END_METHOD

METHOD PUBLIC TestTryDeserializeFrom
VAR
    deserializer : JsonDeserializer;
    feedback : DeserializerFeedback;
    json : STRING(500) := '{"wDay":3,"wDayOfWeek":2,"wHour":4,"wMilliseconds":7,"wMinute":5,"wMonth":1,"wSecond":6,"wYear":2000}';
    _type : _TIMESTRUCT;
    expected : TIMESTRUCT := (wYear := 2000, wMonth := 1, wDayOfWeek := 2, wDay := 3, wHour := 4, wMinute := 5, wSecond := 6, wMilliseconds := 7);
    actual : TIMESTRUCT;
 END_VAR
TEST('TestTryDeserializeFrom');

deserializer.Reset();
deserializer.TryLoad(json);
_type.TryDeserializeFrom(Deserializer, Feedback);

actual := _type.Value;

AssertEquals(
    Expected := expected,
    Actual := actual,
    Message := 'Type did not deserialize correctly.'
);

TEST_FINISHED();
END_METHOD

METHOD PUBLIC TestTryMakeReferenceToFollowsReference
VAR
    _type : _TIMESTRUCT;
	target : _TIMESTRUCT;
    expected : TIMESTRUCT := (wDay := 2);
    actual : TIMESTRUCT;
END_VAR
TEST('TestTryMakeReferenceToFollowsReference');

_type.TryMakeReferenceTo(target);
target.wDay.Value := 2;

actual := _type.Value;

AssertEquals(
    Expected := expected,
    Actual := actual,
    Message := 'Value did not follow target change'
);

TEST_FINISHED();
END_METHOD

METHOD PUBLIC TestTryMakeReferenceToUpdatesReference
VAR
    _type : _TIMESTRUCT;
	target : _TIMESTRUCT;
    expected : TIMESTRUCT := (wDay := 2);
    actual : TIMESTRUCT;
END_VAR
TEST('TestTryMakeReferenceToUpdatesReference');

_type.TryMakeReferenceTo(target);
_type.wDay.Value := 2;

actual := target.Value;

AssertEquals(
    Expected := expected,
    Actual := actual,
    Message := 'Value did not update target'
);

TEST_FINISHED();
END_METHOD

METHOD PUBLIC TestValueReturnsExpectedAfterChange
VAR
    _type : _TIMESTRUCT;
	value : TIMESTRUCT := (wDay := 2);
    expected : TIMESTRUCT := (wDay := 2);
    actual : TIMESTRUCT;
END_VAR
TEST('TestValueReturnsExpectedAfterChange');

_type.Value := value;
actual := _type.Value;

AssertEquals(
    Expected := expected,
    Actual := actual,
    Message := 'Expected value not returned after change.'
);

TEST_FINISHED();
END_METHOD

END_FUNCTION_BLOCK

// ---- Tests/Enums/_E_TcEventClass_TestSuite.TcPOU
FUNCTION_BLOCK _E_TcEventClass_TestSuite EXTENDS TcUnit.FB_TestSuite
VAR
END_VAR

TestAddress();
TestClearReference();
TestClone();
TestIecTypeReturnsExpected();
TestMakeReferenceToFollowsReference();
TestMakeReferenceToUpdatesReference();
TestSize();
TestValueReturnsExpectedAfterInit();
TestValueReturnsExpectedAfterChange();
TestSerializeTypeWith();
TestSerializeWith();
TestTryDeserializeFrom();
TestTryMakeReferenceToFollowsReference();
TestTryMakeReferenceToUpdatesReference();

METHOD PUBLIC TestAddress
VAR
    _type : _E_TcEventClass(E_TcEventClass.TCEVENTCLASS_NONE);
    notExpected : PVOID := 0;
    actual : PVOID;
END_VAR
TEST('TestAddress');

actual := _type.Address;

AssertFalse(
    Condition := (notExpected = actual),
    Message := 'Type did not return a valid address.'
);

TEST_FINISHED();
END_METHOD

METHOD PUBLIC TestClearReference
VAR
    _type : _E_TcEventClass(E_TcEventClass.TCEVENTCLASS_NONE);
	target : E_TcEventClass := E_TcEventClass.TCEVENTCLASS_NONE;
    expected : E_TcEventClass := E_TcEventClass.TCEVENTCLASS_NONE;
    actual : E_TcEventClass;
END_VAR
TEST('TestClearReference');

_type.MakeReferenceTo(target);
_type.ClearReference();
target := E_TcEventClass.TCEVENTCLASS_ALARM;

actual := _type.Value;

AssertEquals(
    Expected := expected,
    Actual := actual,
    Message := 'Value did not follow target change'
);

TEST_FINISHED();
END_METHOD

METHOD PUBLIC TestClone
VAR
    _type : _E_TcEventClass(E_TcEventClass.TCEVENTCLASS_NONE);
	clone : I_Datatype;
	isValidClone : BOOL;
	compareResult : DINT;
END_VAR
TEST('TestClone');

clone := _type.Clone();

isValidClone := clone <> 0;

IF isValidClone THEN
	compareResult := memcmp(_type.Address, clone.Address, clone.Size);
END_IF

AssertTrue(
	Condition := isValidClone,
	Message := 'Clone did not produce a clone'
);

AssertEquals_DINT(
	Expected := 0,
    Actual := compareResult,
    Message := 'Clone did not return a valid clone.'
);

clone.Dispose();

TEST_FINISHED();
END_METHOD

METHOD PUBLIC TestIdentifierReturnsExpected
VAR
    _type : _E_TcEventClass(E_TcEventClass.TCEVENTCLASS_NONE);;
    expected : STRING := 'E_TcEventClass';
    actual : STRING;
END_VAR
TEST('TestIdentifierReturnsExpected');

actual := _type.Identifier;

AssertEquals_STRING(
    Expected := expected,
    Actual := actual,
    Message := 'Type did not return correct iec type.'
);

TEST_FINISHED();
END_METHOD

METHOD PUBLIC TestIecTypeReturnsExpected
VAR
    _type : _E_TcEventClass(E_TcEventClass.TCEVENTCLASS_NONE);;
    expected : STRING := 'ENUM';
    actual : STRING;
END_VAR
TEST('TestIecTypeReturnsExpected');

actual := _type.Datatype;

AssertEquals_STRING(
    Expected := expected,
    Actual := actual,
    Message := 'Type did not return correct iec type.'
);

TEST_FINISHED();
END_METHOD

METHOD PUBLIC TestMakeReferenceToFollowsReference
VAR
    _type : _E_TcEventClass(E_TcEventClass.TCEVENTCLASS_NONE);;
	target : E_TcEventClass := E_TcEventClass.TCEVENTCLASS_NONE;
    expected : E_TcEventClass := E_TcEventClass.TCEVENTCLASS_ALARM;
    actual : E_TcEventClass;
END_VAR
TEST('TestMakeReferenceToFollowsReference');

_type.MakeReferenceTo(target);
target := E_TcEventClass.TCEVENTCLASS_ALARM;

actual := _type.Value;

AssertEquals(
    Expected := expected,
    Actual := actual,
    Message := 'Value did not follow target change'
);

TEST_FINISHED();
END_METHOD

METHOD PUBLIC TestMakeReferenceToUpdatesReference
VAR
    _type : _E_TcEventClass(E_TcEventClass.TCEVENTCLASS_NONE);;
	target : E_TcEventClass := E_TcEventClass.TCEVENTCLASS_NONE;
    expected : E_TcEventClass := E_TcEventClass.TCEVENTCLASS_ALARM;
    actual : E_TcEventClass;
END_VAR
TEST('TestMakeReferenceToUpdatesReference');

_type.MakeReferenceTo(target);
_type.Value := E_TcEventClass.TCEVENTCLASS_ALARM;

actual := target;

AssertEquals(
    Expected := expected,
    Actual := actual,
    Message := 'Value did not update target'
);

TEST_FINISHED();
END_METHOD

METHOD PUBLIC TestSerializeTypeWith
VAR
    _type : _E_TcEventClass(E_TcEventClass.TCEVENTCLASS_NONE);
    serializer : JsonSerializer;
    expected : STRING(500) := '{"datatype":"ENUM","identifier":"E_TcEventClass","enumerations":["TCEVENTCLASS_ALARM","TCEVENTCLASS_HINT","TCEVENTCLASS_INSTRUCTION","TCEVENTCLASS_MAINTENANCE","TCEVENTCLASS_MESSAGE","TCEVENTCLASS_NONE","TCEVENTCLASS_PARAMERROR","TCEVENTCLASS_STATEINFO","TCEVENTCLASS_WARNING"],"baseType":{"datatype":"UINT","lowerBound":0,"upperBound":65535,"isSigned":false}}';
    actual : STRING(500);
END_VAR
TEST('TestSerializeTypeWith');

serializer.Reset();
_type.SerializeTypeWith(serializer);
serializer.TryGetSerializedData(ADR(actual), SIZEOF(actual));

AssertEquals_STRING(
    Expected := expected,
    Actual := actual,
    Message := 'Serialization of type did not return correct string.'
);

TEST_FINISHED();
END_METHOD

METHOD PUBLIC TestSerializeWith
VAR
    _type : _E_TcEventClass(E_TcEventClass.TCEVENTCLASS_ALARM);
    serializer : JsonSerializer;
    expected : STRING := '"TCEVENTCLASS_ALARM"';
    actual : STRING(500);
END_VAR
TEST('TestSerializeWith');

serializer.Reset();
_type.SerializeWith(serializer);
serializer.TryGetSerializedData(ADR(actual), SIZEOF(actual));

AssertEquals_STRING(
    Expected := expected,
    Actual := actual,
    Message := 'Serialization of type data did not return correct string.'
);

TEST_FINISHED();
END_METHOD

METHOD PUBLIC TestSize
VAR
    _type : _E_TcEventClass(E_TcEventClass.TCEVENTCLASS_NONE);;
    expected : UDINT := SIZEOF(E_TcEventClass);
    actual : UDINT;
END_VAR
TEST('TestSize');

actual := _type.Size;

AssertEquals_UDINT(
    Expected := Expected,
    Actual := actual,
    Message := 'Type did not return the correct size.'
);

TEST_FINISHED();
END_METHOD

METHOD PUBLIC TestTryDeserializeFrom
VAR
    deserializer : JsonDeserializer;
    feedback : DeserializerFeedback;
    json : STRING := '"TCEVENTCLASS_ALARM"';
    _type : _E_TcEventClass(E_TcEventClass.TCEVENTCLASS_NONE);
    expected : E_TcEventClass := E_TcEventClass.TCEVENTCLASS_ALARM;
    actual : E_TcEventClass;
 END_VAR
TEST('TestTryDeserializeFrom');

deserializer.Reset();
deserializer.TryLoad(json);
_type.TryDeserializeFrom(Deserializer, Feedback);

actual := _type.Value;

AssertEquals_LREAL(
    Expected := expected,
    Actual := actual,
    Delta := LREAL#0.001,
    Message := 'Type did not deserialize correctly.'
);

TEST_FINISHED();
END_METHOD

METHOD PUBLIC TestTryMakeReferenceToFollowsReference
VAR
    _type : _E_TcEventClass(E_TcEventClass.TCEVENTCLASS_NONE);;
	target : _E_TcEventClass(E_TcEventClass.TCEVENTCLASS_NONE);;
    expected : E_TcEventClass := E_TcEventClass.TCEVENTCLASS_ALARM;
    actual : E_TcEventClass;
END_VAR
TEST('TestTryMakeReferenceToFollowsReference');

_type.TryMakeReferenceTo(target);
target.Value := E_TcEventClass.TCEVENTCLASS_ALARM;

actual := _type.Value;

AssertEquals(
    Expected := expected,
    Actual := actual,
    Message := 'Value did not follow target change'
);

TEST_FINISHED();
END_METHOD

METHOD PUBLIC TestTryMakeReferenceToUpdatesReference
VAR
    _type : _E_TcEventClass(E_TcEventClass.TCEVENTCLASS_NONE);;
	target : _E_TcEventClass(E_TcEventClass.TCEVENTCLASS_NONE);;
    expected : E_TcEventClass := E_TcEventClass.TCEVENTCLASS_ALARM;
    actual : E_TcEventClass;
END_VAR
TEST('TestTryMakeReferenceToUpdatesReference');

_type.TryMakeReferenceTo(target);
_type.Value := E_TcEventClass.TCEVENTCLASS_ALARM;

actual := target.Value;

AssertEquals(
    Expected := expected,
    Actual := actual,
    Message := 'Value did not update target'
);

TEST_FINISHED();
END_METHOD

METHOD PUBLIC TestValueReturnsExpectedAfterChange
VAR
    _type : _E_TcEventClass(E_TcEventClass.TCEVENTCLASS_NONE);;
    expected : E_TcEventClass := E_TcEventClass.TCEVENTCLASS_ALARM;
    actual : E_TcEventClass;
END_VAR
TEST('TestValueReturnsExpectedAfterChange');

_type.Value := E_TcEventClass.TCEVENTCLASS_ALARM;

actual := _type.Value;

AssertEquals(
    Expected := expected,
    Actual := actual,
    Message := 'Expected value not returned after change.'
);

TEST_FINISHED();
END_METHOD

METHOD PUBLIC TestValueReturnsExpectedAfterInit
VAR
    _type : _E_TcEventClass(E_TcEventClass.TCEVENTCLASS_ALARM);
    expected : E_TcEventClass := E_TcEventClass.TCEVENTCLASS_ALARM;
    actual : E_TcEventClass;
END_VAR
TEST('TestValueReturnsExpectedAfterInit');

actual := _type.Value;

AssertEquals(
    Expected := expected,
    Actual := actual,
    Message := 'Expected value not returned after Init.'
);

TEST_FINISHED();
END_METHOD

END_FUNCTION_BLOCK
